{attribute 'no_explicit_call' := 'NormallyClosedSensor is a CLASS and must be accessed using methods or properties'}
FUNCTION_BLOCK NormallyClosedSensor implements I_Sensor
VAR
	input				AT %I*: BOOL;
END_VAR

PROPERTY IsActive : bool
GET
IsActive				:= input;
END_GET
END_PROPERTY

PROPERTY IsNotActive : bool
GET
IsNotActive				:= not input;
END_GET
END_PROPERTY

END_FUNCTION_BLOCK

(* stored: Version 1.1.0.1, ProductVersion 3.1.4024.11
   POU NormallyClosedSensor: Id {f2e2a4e5-2f5d-4474-b654-fc2a4952e61f}, SpecialFunc None
   Property IsActive: Id {2f4e86f3-e2ca-4a94-8db0-f1faab6c85c0}
   Get Get: Id {8bb520cb-35f4-47e0-9c0c-443e850691ac}
   Property IsNotActive: Id {6fe9dfcf-d5e9-4602-bc69-d3d6eef9a674}
   Get Get: Id {ede1b19e-2516-4e88-9541-3be33899d590} *)
